TYPE ST_AutoMode_TransCVCamera :
STRUCT
	Command :ST_CommandBasic;
	Status	:ST_StatusBasic;
	UseBoxCamera	:BOOL;
	BoxCameraDone	:BOOL;
END_STRUCT
END_TYPE

(* stored: Version 1.1.0.1, ProductVersion 3.1.4024.13
   DUT ST_AutoMode_TransCVCamera: Id {d6a01acd-40c1-4fbf-b005-ca20f87d2864} *)
